{attribute 'no_explicit_call' := 'Do not call this POU directly'}
FUNCTION_BLOCK ParentAxis IMPLEMENTS ITF_AxisControl, ITF_CyclicUpdate
VAR
	
	// DO NOT USE DIRECTLY 
	// THIS IS A PARENT CLASS DESIGNED TO PROVIDE A BASE OF KEY VARIABLES / METHODS FOR SUB AXIS CLASSES
	
	_ClassRunningIndicatorToggle	: BOOL;
	
	_LocalState						: INT := 0;
	_InternalCounter				: INT := 0;
	_i								: INT := 0;
	_ErrorCount						: UDINT := 0;
	_CurrentErrorCode				: UDINT := 0;
	_PreviousErrorCode				: UDINT := 0;
	
	
	_IsBusyMoving					: BOOL := FALSE;
	_IsBusyStopping					: BOOL := FALSE;
	_IsReadyForCommand				: BOOL := FALSE;
	_IsDoneWithCommand				: BOOL := FALSE;
	_IsInError						: BOOL := FALSE;
	
	_ErrorRTrig						: R_TRIG;
	
END_VAR

// DO NOT USE DIRECTLY 
// THIS IS A PARENT CLASS DESIGNED TO PROVIDE A BASE OF KEY VARIABLES / METHODS FOR SUB AXIS CLASSES

{attribute 'no_explicit_call' := 'Do not call this METHOD directly'}
METHOD CyclicUpdate : HRESULT
VAR_INPUT
END_VAR
END_METHOD

{attribute 'no_explicit_call' := 'Do not call this METHOD directly'}
METHOD StartDisable : BOOL
StartDisable := TRUE;
RETURN;
END_METHOD

{attribute 'no_explicit_call' := 'Do not call this METHOD directly'}
METHOD StartEnable : BOOL
StartEnable := TRUE;
RETURN;
END_METHOD

{attribute 'no_explicit_call' := 'Do not call this METHOD directly'}
METHOD StartErrorChecking : BOOL
StartErrorChecking := TRUE;
RETURN;
END_METHOD

{attribute 'no_explicit_call' := 'Do not call this METHOD directly'}
METHOD StartMovement : BOOL
StartMovement := TRUE;
RETURN;
END_METHOD

{attribute 'no_explicit_call' := 'Do not call this METHOD directly'}
METHOD StartReset : BOOL
StartReset := TRUE;
RETURN;
END_METHOD

END_FUNCTION_BLOCK

(* stored: Version 1.1.0.1, ProductVersion 3.1.4024.12
   POU ParentAxis: Id {819c0fc3-3048-4b65-9596-1ddff471cc22}, SpecialFunc None
   Folder METH: Id {9065e467-db2a-4ff1-919c-a2bed8632ec4}
   Folder PROP: Id {8f4b04f3-ce15-4083-bfcd-af944ad40776}
   Method CyclicUpdate: Id {a76f7c7e-e079-4023-9fb3-ec0d922c9bf3}
   Method StartDisable: Id {56eb439f-d18d-4390-8764-08abcc7c06b0}
   Method StartEnable: Id {16a0593b-8451-40d9-aee4-d72a0c9450e4}
   Method StartErrorChecking: Id {e099fb98-62c2-4bb2-bb4b-4d2033d38bd7}
   Method StartMovement: Id {c1b941a6-8c20-4d78-95eb-da6a932feb1a}
   Method StartReset: Id {814fd21e-0534-46a5-96f8-965c297e8abe} *)
